SUBAPPLICATION mapping_DataPanel (* Subapplication Type *)
  (* Standard: 61499-2 *)
  (* Version 1.0, 2023-01-29, Franz *)
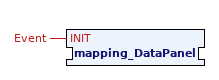
  EVENT_INPUT
    INIT;
  END_EVENT
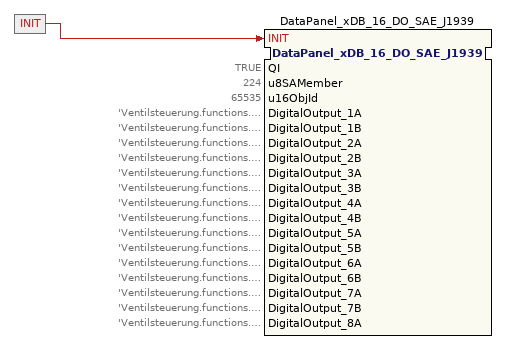
  FBS
    DataPanel_xDB_16_DO_SAE_J1939 : DataPanel_xDB_16_DO_SAE_J1939(QI := TRUE, u8SAMember := 224, u16ObjId := 65535, DigitalOutput_1A := 'Ventilsteuerung.functions.Schneidwerk.rechtslauf', DigitalOutput_1B := 'Ventilsteuerung.functions.Schneidwerk.linkslauf', DigitalOutput_2A := 'Ventilsteuerung.functions.Vorsteuerventil_2A.QX', DigitalOutput_2B := 'Ventilsteuerung.functions.Vorsteuerventil_2B.QX', DigitalOutput_3A := 'Ventilsteuerung.functions.Klappen.Sitzventile.QXA', DigitalOutput_3B := 'Ventilsteuerung.functions.Klappen.Sitzventile.QXB', DigitalOutput_4A := 'Ventilsteuerung.functions.Verteiler.Sitzventile.QXA', DigitalOutput_4B := 'Ventilsteuerung.functions.Verteiler.Sitzventile.QXB', DigitalOutput_5A := 'Ventilsteuerung.functions.Knickdeichsel.Sitzventile.QXA', DigitalOutput_5B := 'Ventilsteuerung.functions.Knickdeichsel.Sitzventile.QXB', DigitalOutput_6A := 'Ventilsteuerung.functions.Dom.QX', DigitalOutput_6B := 'Ventilsteuerung.functions.Heckschieber.QXB', DigitalOutput_7A := 'Ventilsteuerung.functions.Seitenschieber.QX', DigitalOutput_7B := 'Ventilsteuerung.functions.Abscheider.QX', DigitalOutput_8A := 'Ventilsteuerung.functions.Licht.QX');
  END_FBS
  EVENT_CONNECTIONS
    INIT TO DataPanel_xDB_16_DO_SAE_J1939.INIT;
  END_CONNECTIONS
END_SUBAPPLICATION
